FUNCTION_BLOCK logiBUS_IB (* Input service interface function block for byte input data *)
  (* Description: Copyright (c) 2018 TU Wien/ACIN, HR Agrartechnik GmbH This program and the accompanying materials are made available under the terms of the Eclipse Public License 2.0 which is available at https://www.eclipse.org/legal/epl-2.0/ SPDX-License-Identifier: EPL-2.0 this works for: BUTTON_PRESS_REPEAT BUTTON_PRESS_REPEAT_DONE *)
  (* Version 1.0, 2018-10-05, Martin Melik-Merkumians, TU Wien/ACIN, initial API and implementation and/or initial documentation *)
  PACKAGE logiBUS::io::DI;
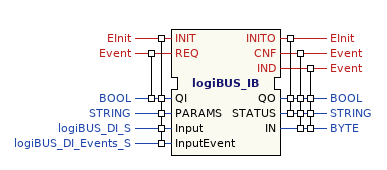
  EVENT_INPUT
    INIT : EInit WITH QI, PARAMS, Input, InputEvent; (* Service Initialization *)
    REQ WITH QI; (* Service Request *)
  END_EVENT
  EVENT_OUTPUT
    INITO : EInit WITH QO, STATUS; (* Initialization Confirm *)
    CNF WITH QO, STATUS, IN; (* Confirmation of Requested Service *)
    IND WITH QO, STATUS, IN; (* Indication from Resource *)
  END_EVENT
  VAR_INPUT
    QI : BOOL; (* Event Input Qualifier *)
    PARAMS : STRING; (* Service Parameters *)
    Input : logiBUS::io::DI::logiBUS_DI_S := logiBUS_DI::Invalid; (* Identify the Input Input_I1..I8 *)
    InputEvent : logiBUS::io::DI::logiBUS_DI_Events_S := logiBUS_DI_Events::Invalid; (* Identify the Event (currently only REPEAT supported) *)
  END_VAR
  VAR_OUTPUT
    QO : BOOL; (* Event Output Qualifier *)
    STATUS : STRING; (* Service Status *)
    IN : BYTE; (* Input data from resource *)
  END_VAR
END_FUNCTION_BLOCK
